DEVICE_TYPE RMT_DEV3 (* Subclass of RMT_DEV *)
  (* Standard: 61499-2 *)
  (* Version 0.2, 2003-12-05, JHC, Rockwell Automation, Renamed from NEWDEVICE. *)
  (* Version 0.1, 2002-11-05, JHC, Rockwell Automation, Corrected <DeviceFBNetwork> to <FBNetwork>. *)
  (* Version 0.0, 2000-05-27, JHC, Rockwell Automation *)
  (* Compiler header: import fb.rt.ita.*; import fb.rt.math.*; *)
  (* Compiler classdef: public class RMT_DEV3 extends FBDevice implements RemoteDevice *)
  RESOURCE RES1 : EMB_RES2
  END_RESOURCE
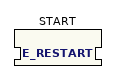
  FBS
    START : E_RESTART;
  END_FBS
END_DEVICE_TYPE
